FUNCTION FC_DistMod : LREAL
VAR_INPUT
	fPosFrom:LREAL;
	fPosTo:LREAL;
	fModRange:LREAL;
END_VAR
VAR
	fDist:LREAL;
	fDist1:LREAL;
END_VAR

  // check closest direction between two points

IF fPosTo > fPosFrom THEN
  IF fPosTo - fPosFrom < 360 - fPosTo+ fPosFrom THEN
    fDist:=fPosTo - fPosFrom;  //forward
  ELSE	
    fDist:=-( 360 - fPosTo+ fPosFrom);  //backward
  END_IF
ELSE
  IF fPosFrom - fPosTo < fPosTo + 360 - fPosFrom THEN
	fDist:=-(fPosFrom - fPosTo); //Backward
  ELSE	
    fDist:=fPosTo + 360 - fPosFrom;  //Forward
  END_IF
END_IF

FC_DistMod:= fDist;

END_FUNCTION

(* stored: Version 1.1.0.1, ProductVersion 3.1.4024.6
   POU FC_DistMod: Id {ab909bcd-5527-41a8-a57f-59891c5d6be4}, SpecialFunc None *)
